// TIA Portal V20 export
DATA_BLOCK "PM7"   // DB281
// stored: MemoryReserve 100
   VAR
      SPARE : Bool;
      SPARE_1 : Bool;
      SPARE_2 : Bool;
      SPARE_3 : Bool;
      SPARE_4 : Bool;
      SPARE_5 : Bool;
      SPARE_6 : Bool;
      SPARE_7 : Bool;
      "HP STAGE LIFT #1 FRONT UP" : Bool;
      "HP STAGE LIFT #1 FRONT DOWN" : Bool;
      "HP STAGE LIFT #1 REAR UP" : Bool;
      "HP STAGE LIFT #1 REAR DOWN" : Bool;
      "HP STAGE LIFT #2 FRONT UP" : Bool;
      "HP STAGE LIFT #2 FRONT DOWN" : Bool;
      "HP STAGE LIFT #2 REAR UP" : Bool;
      "HP STAGE LIFT #2 REAR DOWN" : Bool;
   END_VAR
BEGIN
END_DATA_BLOCK
